(*

.. <legal notes>

legal notes
=================
| SPDX-FileCopyrightText: © 2026 Oleksandr Tiutyk <trofimich@gmail.com>
| SPDX-License-Identifier: LGPL-3.0-only
| For details check: LGPL-3.0-only_

.. _LGPL-3.0-only: https://www.gnu.org/licenses/lgpl-3.0.en.html

.. </legal notes>

*)

INTERFACE IDynamicByteList EXTENDS IReadOnlyDynamicByteList

METHOD AppendAny : IDynamicByteList
VAR_INPUT
	data : ANY;
END_VAR
END_METHOD

METHOD AppendByte : IDynamicByteList
VAR_INPUT
	value : BYTE;
END_VAR
END_METHOD

METHOD AppendData : IDynamicByteList
VAR_INPUT
	data : POINTER TO BYTE;
	dataSize : UDINT;
END_VAR
END_METHOD

METHOD AppendGeneric : IDynamicByteList
VAR_INPUT
	data : Core.GENERIC_VALUE;
END_VAR
END_METHOD

METHOD Clear : IDynamicByteList
VAR_INPUT
	releaseMemory : BOOL := FALSE;
END_VAR
END_METHOD

METHOD LoadFromAny : IDynamicByteList
VAR_INPUT
	data : ANY;
	startIndex : COLLECTION_INDEX := 0;
END_VAR
END_METHOD

METHOD LoadFromData : IDynamicByteList
VAR_INPUT
	data : POINTER TO BYTE;
	dataSize : ULINT;
	startIndex : COLLECTION_INDEX := 0;
END_VAR
END_METHOD

METHOD LoadFromGeneric : IDynamicByteList
VAR_INPUT
	data : Core.GENERIC_VALUE;
	startIndex : COLLECTION_INDEX := 0;
END_VAR
END_METHOD

METHOD Remove : IDynamicByteList
VAR_INPUT
	value : BYTE;
END_VAR
END_METHOD

METHOD RemoveAt : IDynamicByteList
VAR_INPUT
	index : COLLECTION_INDEX;
	count : COLLECTION_LENGTH := 1;
END_VAR
END_METHOD

METHOD Resize : IDynamicByteList
VAR_INPUT
	newBytesCount : DINT;
END_VAR
END_METHOD

METHOD Set : IDynamicByteList
VAR_INPUT
	index : COLLECTION_INDEX;
	value : BYTE;
END_VAR
END_METHOD

END_INTERFACE

(* stored: Version 1.1.0.1
   Itf IDynamicByteList: Id {518eb55c-df07-0206-0227-e692a273d945}
   Method AppendAny: Id {1b640082-c494-4770-8a43-3eb7addbc09e}
   Method AppendByte: Id {1ab7d3cb-0dd2-4a95-871a-2df749dcb5a5}
   Method AppendData: Id {1186b88b-e5f6-4d0a-850c-7b49aca8e28d}
   Method AppendGeneric: Id {c20b42af-40c5-495e-b096-4ffb90d5ad93}
   Method Clear: Id {243fdc07-7928-4ca7-a298-f89f02bbd736}
   Method LoadFromAny: Id {b3c42220-f6d9-4c15-b9b4-e89b6fac55f8}
   Method LoadFromData: Id {f1c6da5c-ced0-42ee-9f57-c45302a7ebcb}
   Method LoadFromGeneric: Id {0e129b3d-d8f7-4a58-8e16-3c8b5d4146dc}
   Method Remove: Id {eed9e02a-e972-481f-8ddf-d0d8fccc576a}
   Method RemoveAt: Id {5d545c6c-7499-43af-8e59-315db670ead5}
   Method Resize: Id {c4504f91-d8a1-4fc4-bf4f-18aa14caa2ad}
   Method Set: Id {267c54d8-2df6-0ce5-162c-03537dc39a04} *)
